(*

short summary
=================
This interface provides assert statements for windows-1252 strings until 255 characters length

.. <legal notes>

legal notes
=================
| SPDX-FileCopyrightText: © 2022 ekvip automation GmbH <info@ekvip.de>
| SPDX-License-Identifier: Apache-2.0
| For details check: Apache-2.0_

.. _Apache-2.0: https://www.apache.org/licenses/LICENSE-2.0

.. </legal notes>

methods
==================

*)

INTERFACE IWindows1252StringAssertions EXTENDS __SYSTEM.IQueryInterface

(*

short summary
=================
This assertion method checks if the current string ``stringToCheck`` contains the search string

.. <legal notes>

legal notes
=================
| SPDX-FileCopyrightText: © 2022 ekvip automation GmbH <info@ekvip.de>
| SPDX-License-Identifier: Apache-2.0
| For details check: Apache-2.0_

.. _Apache-2.0: https://www.apache.org/licenses/LICENSE-2.0

.. </legal notes>

parameters
=================

*)

METHOD contains
VAR_INPUT
	(* current string to check *)
	stringToCheck	:Tc2_System.T_MaxString;
	(* string must be found in ``stringToCheck`` *)
	searchString	:Tc2_System.T_MaxString;
	(* ``TRUE`` means ignore cases; ``FALSE`` means cases must be equal too *)
	ignoreCases		:BOOL;
	(* message if the assertion is false *)
	message			:AssertMessage;
END_VAR
END_METHOD

(*

short summary
=================
This assertion method checks if the current string ``stringToCheck`` not contains the search string

.. <legal notes>

legal notes
=================
| SPDX-FileCopyrightText: © 2022 ekvip automation GmbH <info@ekvip.de>
| SPDX-License-Identifier: Apache-2.0
| For details check: Apache-2.0_

.. _Apache-2.0: https://www.apache.org/licenses/LICENSE-2.0

.. </legal notes>

parameters
=================

*)

METHOD containsNo
VAR_INPUT
	(* current string to check *)
	stringToCheck	:Tc2_System.T_MaxString;
	(* string that must not be found in ``stringToCheck`` *)
	searchString	:Tc2_System.T_MaxString;
	(* ``TRUE`` means ignore cases; ``FALSE`` means cases must be equal too *)
	ignoreCases		:BOOL;
	(* message if the assertion is false *)
	message			:AssertMessage;
END_VAR
END_METHOD

(*

short summary
=================
This assertion method checks if the current string ``stringToCheck`` ends with ``end``

.. <legal notes>

legal notes
=================
| SPDX-FileCopyrightText: © 2022 ekvip automation GmbH <info@ekvip.de>
| SPDX-License-Identifier: Apache-2.0
| For details check: Apache-2.0_

.. _Apache-2.0: https://www.apache.org/licenses/LICENSE-2.0

.. </legal notes>

parameters
=================

*)

METHOD endsWith
VAR_INPUT
	(* current string to check *)
	stringToCheck	:Tc2_System.T_MaxString;
	(* expected end of ``stringToCheck`` *)
	end				:Tc2_System.T_MaxString;
	(* ``TRUE`` means ignore cases; ``FALSE`` means cases must be equal too *)
	ignoreCases		:BOOL;
	(* ``TRUE`` means truncation of spaces on the right side of ``stringToCheck``*)
	trim			:BOOL;
	(* message if the assertion is false *)
	message			:AssertMessage;
END_VAR
END_METHOD

(*

short summary
=================
This assertion method checks if the current string ``stringToCheck`` is empty

.. <legal notes>

legal notes
=================
| SPDX-FileCopyrightText: © 2022 ekvip automation GmbH <info@ekvip.de>
| SPDX-License-Identifier: Apache-2.0
| For details check: Apache-2.0_

.. _Apache-2.0: https://www.apache.org/licenses/LICENSE-2.0

.. </legal notes>

parameters
=================

*)

METHOD isEmpty
VAR_INPUT
	(* current string to check *)
	stringToCheck	:Tc2_System.T_MaxString;
	(* message if the assertion is false *)
	message			:AssertMessage;
END_VAR
END_METHOD

(*

short summary
=================
This assertion method checks if the current string ``stringToCheck`` is equal to ``expected``

.. <legal notes>

legal notes
=================
| SPDX-FileCopyrightText: © 2022 ekvip automation GmbH <info@ekvip.de>
| SPDX-License-Identifier: Apache-2.0
| For details check: Apache-2.0_

.. _Apache-2.0: https://www.apache.org/licenses/LICENSE-2.0

.. </legal notes>

parameters
=================

*)

METHOD isEqualTo
VAR_INPUT
	(* current string to check *)
	stringToCheck	:Tc2_System.T_MaxString;
	(* ``stringToCheck`` must be equal to expected *)
	expected		:Tc2_System.T_MaxString;
	(* ``TRUE`` means ignore cases; ``FALSE`` means cases must be equal too *)
	ignoreCases		:BOOL;
	(* message if the assertion is false *)
	message			:AssertMessage;
END_VAR
END_METHOD

(*

short summary
=================
This assertion method checks if the current string ``stringToCheck`` is not empty

.. <legal notes>

legal notes
=================
| SPDX-FileCopyrightText: © 2022 ekvip automation GmbH <info@ekvip.de>
| SPDX-License-Identifier: Apache-2.0
| For details check: Apache-2.0_

.. _Apache-2.0: https://www.apache.org/licenses/LICENSE-2.0

.. </legal notes>

parameters
=================

*)

METHOD isNotEmpty
VAR_INPUT
	(* current string to check *)
	stringToCheck	:Tc2_System.T_MaxString;
	(* message if the assertion is false *)
	message			:AssertMessage;
END_VAR
END_METHOD

(*

short summary
=================
This assertion method checks if the current string ``stringToCheck`` is not equal to ``unexpected``

.. <legal notes>

legal notes
=================
| SPDX-FileCopyrightText: © 2022 ekvip automation GmbH <info@ekvip.de>
| SPDX-License-Identifier: Apache-2.0
| For details check: Apache-2.0_

.. _Apache-2.0: https://www.apache.org/licenses/LICENSE-2.0

.. </legal notes>

parameters
=================

*)

METHOD isNotEqualTo
VAR_INPUT
	(* current string to check *)
	stringToCheck	:Tc2_System.T_MaxString;
	(* ``stringToCheck`` must be not equal to expected *)
	unexpected		:Tc2_System.T_MaxString;
	(* ``TRUE`` means ignore cases; ``FALSE`` means cases must be equal too *)
	ignoreCases		:BOOL;
	(* message if the assertion is false *)
	message			:AssertMessage;
END_VAR
END_METHOD

(*

short summary
=================
This assertion method checks if the current string ``stringToCheck`` is length
is between ``minLenght`` and ``maxLenght``

.. <legal notes>

legal notes
=================
| SPDX-FileCopyrightText: © 2022 ekvip automation GmbH <info@ekvip.de>
| SPDX-License-Identifier: Apache-2.0
| For details check: Apache-2.0_

.. _Apache-2.0: https://www.apache.org/licenses/LICENSE-2.0

.. </legal notes>

parameters
=================

*)

METHOD lenghtIsBetween
VAR_INPUT
	(* current string to check *)
	stringToCheck	:Tc2_System.T_MaxString;
	(* lower limit of the string length *)
	minLenght	:USINT;
	(* upper limit of the string length *)
	maxLenght	:USINT;
	(* message if the assertion is false *)
	message			:AssertMessage;
END_VAR
END_METHOD

(*

short summary
=================
This assertion method checks if the current string ``stringToCheck`` is length
is equal to ``expectedLength``

.. <legal notes>

legal notes
=================
| SPDX-FileCopyrightText: © 2022 ekvip automation GmbH <info@ekvip.de>
| SPDX-License-Identifier: Apache-2.0
| For details check: Apache-2.0_

.. _Apache-2.0: https://www.apache.org/licenses/LICENSE-2.0

.. </legal notes>

parameters
=================

*)

METHOD lenghtIsExact
VAR_INPUT
	(* current string to check *)
	stringToCheck	:Tc2_System.T_MaxString;
	(* expected length of ``stringToCheck`` *)
	expectedLength	:USINT;
	(* message if the assertion is false *)
	message			:AssertMessage;
END_VAR
END_METHOD

(*

short summary
=================
This assertion method checks if the current string ``stringToCheck`` is length
is equal or less than to ``maxLength``

.. <legal notes>

legal notes
=================
| SPDX-FileCopyrightText: © 2022 ekvip automation GmbH <info@ekvip.de>
| SPDX-License-Identifier: Apache-2.0
| For details check: Apache-2.0_

.. _Apache-2.0: https://www.apache.org/licenses/LICENSE-2.0

.. </legal notes>

parameters
=================

*)

METHOD lenghtIsMax
VAR_INPUT
	(* current string to check *)
	stringToCheck	:Tc2_System.T_MaxString;
	(* upper limit of the length of ``stringToCheck`` *)
	maxLength		:USINT;
	(* message if the assertion is false *)
	message			:AssertMessage;
END_VAR
END_METHOD

(*

short summary
=================
This assertion method checks if the current string ``stringToCheck`` is length
is equal or grater than to ``minLength``

.. <legal notes>

legal notes
=================
| SPDX-FileCopyrightText: © 2022 ekvip automation GmbH <info@ekvip.de>
| SPDX-License-Identifier: Apache-2.0
| For details check: Apache-2.0_

.. _Apache-2.0: https://www.apache.org/licenses/LICENSE-2.0

.. </legal notes>

parameters
=================

*)

METHOD lenghtIsMin
VAR_INPUT
	(* current string to check *)
	stringToCheck	:Tc2_System.T_MaxString;
	(* lower limit of the length of ``stringToCheck`` *)
	minLength	:USINT;
	(* message if the assertion is false *)
	message			:AssertMessage;
END_VAR
END_METHOD

(*

short summary
=================
This assertion method checks if the current string ``stringToCheck`` starts with ``start``

.. <legal notes>

legal notes
=================
| SPDX-FileCopyrightText: © 2022 ekvip automation GmbH <info@ekvip.de>
| SPDX-License-Identifier: Apache-2.0
| For details check: Apache-2.0_

.. _Apache-2.0: https://www.apache.org/licenses/LICENSE-2.0

.. </legal notes>

parameters
=================

*)

METHOD startsWith
VAR_INPUT
	(* current string to check *)
	stringToCheck	:Tc2_System.T_MaxString;
	(* expected start of ``stringToCheck`` *)
	start			:Tc2_System.T_MaxString;
	(* ``TRUE`` means ignore cases; ``FALSE`` means cases must be equal too *)
	ignoreCases		:BOOL;
	(* ``TRUE`` means truncation of spaces on the left side of ``stringToCheck``*)
	trim			:BOOL;
	(* message if the assertion is false *)
	message			:AssertMessage;
END_VAR
END_METHOD

END_INTERFACE

(* stored: Version 1.1.0.1, ProductVersion 3.1.4024.12
   Itf IWindows1252StringAssertions: Id {fc4f0a8e-4a45-4b9e-b1f7-dcf5428de708}
   Method contains: Id {9eb17bd8-b417-4a97-a78b-bb8671a3deb5}
   Method containsNo: Id {b6b2dea8-ff13-46d1-bd20-7ece860d922d}
   Method endsWith: Id {5f1e09d7-e7dc-45bf-8913-198e3bad95c4}
   Method isEmpty: Id {e68800b8-8a0f-4587-981b-d3f0ee280058}
   Method isEqualTo: Id {a2643ecc-4952-4138-a2d1-aa531444c798}
   Method isNotEmpty: Id {c9dbac78-e03c-4a32-8025-60757c1060a1}
   Method isNotEqualTo: Id {64d22111-a99f-4bbd-b39a-27bd32351861}
   Method lenghtIsBetween: Id {5508718c-8aef-4252-8a69-b1618b40428e}
   Method lenghtIsExact: Id {fed3fe4d-9a2a-43ba-9fe5-7598efb817e3}
   Method lenghtIsMax: Id {c7f179db-bc83-4c4a-ac27-d23f06084900}
   Method lenghtIsMin: Id {ae0d7497-b215-4cc5-9710-119eec82cbdb}
   Method startsWith: Id {56973902-a8c9-4eab-820e-bcf13e55ded4} *)
